PROGRAM SYSTEM
VAR
END_VAR

HMI_Global.fbGetLocalSystemTime(
	sNetID:= , 
	bEnable:= TRUE, 
	dwCycle:= 1, 
	dwOpt:= , 
	tTimeout:= , 
	bValid=> , 
	systemTime=> , 
	tzID=> );
	
HMI_Global.sSystemDateTime := SYSTEMTIME_TO_STRING(HMI_Global.fbGetLocalSystemTime.systemTime);
HMI_Global.sSystemDate := MID(STR:= HMI_Global.sSystemDateTime, LEN:=10, POS:=1);
HMI_Global.sSystemTime := MID(STR:= HMI_Global.sSystemDateTime, LEN:=8, POS:=12);

END_PROGRAM

(* stored: Version 1.1.0.1, ProductVersion 3.1.4024.12
   POU SYSTEM: Id {ec2b8c0a-e8a6-4c50-8d63-8b8bda8e76b5}, SpecialFunc None *)
